FUNCTION_BLOCK IN_ENUM (* Enumerated data input from drop-down list *)
  (* Standard: 61499-1; Classification: GUI *)
  (* Version 0.4, 2006-03-19, JHC, Holobloc Inc, Changed package to fb.rt.hmi *)
  (* Version 0.3, 2004-06-21, JHC, Rockwell Automation, Made composite, Swing implementation. *)
  (* Version 0.2, 2002-05-03, JHC, Rockwell Automation, Made QI IV=true. *)
  (* Version 0.1, 2001-06-08, JHC, Rockwell Automation, XML version, concrete *)
  (* Version 0.0, 1998-11-20, JHC, Rockwell Automation, Original (Java) version, abstract *)
  (* Compiler header: package fb.rt.hmi; *)
  (* Compiler Java Sun JDK 1.4.2 *)
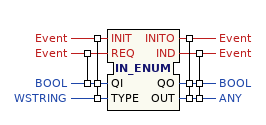
  EVENT_INPUT
    INIT WITH QI, TYPE;
    REQ WITH QI;
  END_EVENT
  EVENT_OUTPUT
    INITO WITH QO, OUT;
    IND WITH QO, OUT;
  END_EVENT
  VAR_INPUT
    QI : BOOL := true;
    TYPE : WSTRING := "ANY"; (* Data type name,must be enumerated type *)
  END_VAR
  VAR_OUTPUT
    QO : BOOL; (* 1=OK,0=Error *)
    OUT : ANY;
  END_VAR
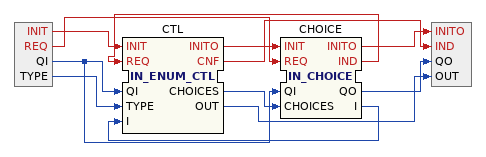
  FBS
    CHOICE : IN_CHOICE;
    CTL : IN_ENUM_CTL;
  END_FBS
  EVENT_CONNECTIONS
    INIT TO CTL.INIT;
    CTL.INITO TO CHOICE.INIT;
    CHOICE.INITO TO INITO;
    REQ TO CHOICE.REQ;
    CHOICE.IND TO CTL.REQ;
    CTL.CNF TO IND;
  END_CONNECTIONS
  DATA_CONNECTIONS
    QI TO CTL.QI;
    QI TO CHOICE.QI;
    CHOICE.QO TO QO;
    TYPE TO CTL.TYPE;
    CTL.CHOICES TO CHOICE.CHOICES;
    CHOICE.I TO CTL.I;
    CTL.OUT TO OUT;
  END_CONNECTIONS
END_FUNCTION_BLOCK
